FUNCTION_BLOCK INTERNAL FINAL SignalListExtender
VAR
	_iList		: I_SignalList;
END_VAR

PROPERTY INTERNAL List : I_SignalList
GET
List := _iList;
END_GET
SET
_iList := List;
END_SET
END_PROPERTY

END_FUNCTION_BLOCK

(* stored: Version 1.1.0.1
   POU SignalListExtender: Id {0f799782-1ff9-4e36-a7c9-b4588827fc12}, SpecialFunc None
   Property List: Id {487fe7c7-f5f3-47a8-bafe-6491cdde4457}
   Get Get: Id {f0efffd7-2c40-4e68-8922-fe371c28bca9}
   Set Set: Id {f376151b-771b-46cd-81e9-5b7a4fcdaaab} *)
